		IF iObjState = 1 THEN																							// Objekt wurde geresettet
			iSkillCommand := 0;																								// Zurücksetzen von Command
			bDone := FALSE;																									// Zurücksetzen von Skill
			bSkillFertig := TRUE;									
		END_IF
			
		//  TRANSITION
		IF bSkillFertig THEN
			bSkillFertig := FALSE;																																											// Resetten von Objekt
			iState := 0;
		END_IF
		
// _________________________________________________________________________________________________________________________
3: 	// FEHLER
		// DO 	
		iSkillCommand := 0;
		
		bDone := FALSE;
		bBusy := FALSE;
		
		// TRANSITION
		IF bResetten THEN
			iState := 0;
		END_IF
		
// _________________________________________________________________________________________________________________________			
4: 	// LIMIT
		// DO 
		iSkillCommand := 0;
		bLimit := TRUE;																									// Limit wurde erreicht
		
		iSkillCommand := 3;																								// Objekt resetten
		
		IF iObjState = 1 THEN																							// Objekt wurde geresettet
			iSkillCommand := 0;																								// Zurücksetzen von Command
			bDone := FALSE;																									// Zurücksetzen von Skill
			bResetten := TRUE;								
		END_IF
	
		// TRANSITION
		IF bResetten THEN
			bResetten := FALSE;
			bLimit := FALSE;																							// Zurücksetzen von Output-Variable
			iSkillCommand := 3;																							// Resetten von Objekt 
			iState := 0;
		END_IF
			
// _________________________________________________________________________________________________________________________
5: 	// ERREICHT		
		// DO 
		iSkillCommand := 0;
		bDone := TRUE;																									// Skill wurde erfolgreich ausgeführt
		
		iSkillCommand := 3;																								// Objekt resetten
		
		IF iObjState = 1 THEN																							// Objekt wurde geresettet
			iSkillCommand := 0;																								// Zurücksetzen von Command
			bDone := FALSE;																									// Zurücksetzen von Skill
			bSkillFertig := TRUE;									
		END_IF
		
		// TRANSITION
		IF bSkillFertig THEN
			bSkillFertig := FALSE;
			iState := 0;
		END_IF
		
END_CASE

END_FUNCTION_BLOCK

// ---- POUs/01_Prozessmodell/02_Sequenzen/Seq_1.TcPOU
FUNCTION_BLOCK Seq_1
VAR_INPUT
	// Basis-Inputs
	bExecute			:BOOL;				// Trigger für Ausführung von Sequenz
	iSysCommand			:eSystemCommand;	// Steuerungsvariabel von System (Resetten)
	iSysState			:eSystemState;		// Information über Zustand von System
	
	
	// Prozess-Inputs 
	Position_1			:sRoboterProzessVariablen;
	Position_DOWN		:sRoboterProzessVariablen;
	Position_UP			:sRoboterProzessVariablen;
	Position_2			:sRoboterProzessVariablen;
END_VAR
VAR_OUTPUT
	bDone				:BOOL;				// Information ob Sequenz ausgfeührt wurde
	bBusy				:BOOL;				// Information ob Sequenz im Moment ausgeführt wird
	bError				:BOOL;				// Information ob sich Sequenz in Fehlerzustand befindet
END_VAR
VAR
	// Sequenz-Zustände
	iState				:eSequenceState;
	
	// Startvariablen (FB soll nur bei einer steigenden Flanke gestartet werden)
	fTrigger			:R_TRIG;			// Erkennung einer steigenden Flanke für den Starte
	fSwitch				:SR;				// Setzen des Signals
	bSwitchResett		:BOOL;				// Resetten des Signals
	
	// Zustandsvariablen
	bStarten			:BOOL;
	bStoppen			:BOOL;
	bResetten			:BOOL;
	
	// Management-Variablen:
	bFinished			:BOOL;
	bInit				:BOOL;
	
	// Skill-Instanziierungen
	P2P_Bewegung		:Skill_Position_anfahren;
	Position			:sRoboterProzessVariablen;
	
END_VAR

// Aufrufen von Skills und Ablauf
Ablauf();	
Skills();

//_______________________________________________________________
// Reaktion auf Fehler
IF bError THEN
	iState := 3;
END_IF	

// Reaktion auf Input-Variablen: 
	// Starten
	fTrigger(CLK := bExecute);
	fSwitch(Set1 := fTrigger.Q);
	
	IF fSwitch.Q1 THEN
		bStarten := TRUE;
	ELSE
		bStarten := FALSE;
	END_IF
	
	// Stoppen
	IF iSysCommand = 3 THEN
		bStoppen := TRUE;	
	ELSE 
		bStoppen := FALSE;	
	END_IF
	
	// Stoppen
	IF iSysCommand = 4 THEN
		bResetten := TRUE;	
	ELSE 
		bResetten := FALSE;	
	END_IF



//_______________________________________________________________
// Zustandsmanagement
CASE iState OF 
	0:	// BEREIT
			// DO	
			fSwitch.RESET := FALSE;
				
			// TRANSITION
			IF bStarten THEN
				fSwitch.RESET := TRUE;
				iState := 1;																							// Starten des Objektes 
			END_IF
	// ________________________________________________________________________________			
	1:	// LAUFEND
			// DO
			bBusy := TRUE;	

			IF bStoppen THEN
				SFCReset := TRUE;
				bBusy := FALSE;
			END_IF	
			
			// TRANSITION
			IF bFinished THEN
				bFinished := FALSE;
				bBusy := FALSE;
				iState := 2;
			END_IF
			
			IF bInit THEN
				bInit := FALSE;
				SFCReset := FALSE;
				iState := 0;
			END_IF

	// ________________________________________________________________________________					
	2:	// ABGESCHLOSSEN
			// DO
			bDone := TRUE;			
						
			// TRANSITION
			IF bDone THEN
				bDone := FALSE;
				iState := 0;
			END_IF
	// ________________________________________________________________________________					
	3:	// FEHLER
			// DO
			bDone := FALSE;
			bBusy := FALSE;
			
			// TRANSITION
			IF bResetten THEN
				bError := FALSE;
				iState := 0;
			END_IF
			
END_CASE

ACTION Ablauf:
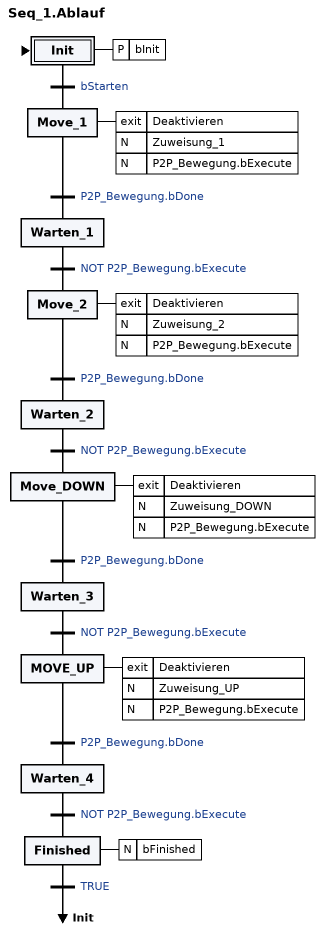
INITIAL_STEP Init:
    bInit(P);
END_STEP
TRANSITION FROM Init TO Move_1
    := bStarten;
END_TRANSITION
STEP Move_1:
    Deaktivieren(P0);  // exit action
    Zuweisung_1(N);
    P2P_Bewegung.bExecute(N);
END_STEP
TRANSITION FROM Move_1 TO Warten_1
    := P2P_Bewegung.bDone;
END_TRANSITION
STEP Warten_1:
END_STEP
TRANSITION FROM Warten_1 TO Move_2
    := NOT P2P_Bewegung.bExecute;
END_TRANSITION
STEP Move_2:
    Deaktivieren(P0);  // exit action
    Zuweisung_2(N);
    P2P_Bewegung.bExecute(N);
END_STEP
TRANSITION FROM Move_2 TO Warten_2
    := P2P_Bewegung.bDone;
END_TRANSITION
STEP Warten_2:
END_STEP
TRANSITION FROM Warten_2 TO Move_DOWN
    := NOT P2P_Bewegung.bExecute;
END_TRANSITION
STEP Move_DOWN:
    Deaktivieren(P0);  // exit action
    Zuweisung_DOWN(N);
    P2P_Bewegung.bExecute(N);
END_STEP
TRANSITION FROM Move_DOWN TO Warten_3
    := P2P_Bewegung.bDone;
END_TRANSITION
STEP Warten_3:
END_STEP
TRANSITION FROM Warten_3 TO MOVE_UP
    := NOT P2P_Bewegung.bExecute;
END_TRANSITION
STEP MOVE_UP:
    Deaktivieren(P0);  // exit action
    Zuweisung_UP(N);
    P2P_Bewegung.bExecute(N);
END_STEP
TRANSITION FROM MOVE_UP TO Warten_4
    := P2P_Bewegung.bDone;
END_TRANSITION
STEP Warten_4:
END_STEP
TRANSITION FROM Warten_4 TO Finished
    := NOT P2P_Bewegung.bExecute;
END_TRANSITION
STEP Finished:
    bFinished(N);
END_STEP
TRANSITION FROM Finished TO Init
    := TRUE;
END_TRANSITION
END_ACTION

ACTION Deaktivieren:
P2P_Bewegung.bExecute := FALSE;
END_ACTION

ACTION Skills:
P2P_Bewegung(
    iSysCommand := GVL.SystemCommand,
    iObjState := Anlage.UR5.P_State,
    iSysState := GVL.SystemState,
    sProzessvariablen := Position); // Skill_Position_anfahren
Anlage.UR5.Prozessvariablen := P2P_Bewegung.sObjektvariablen;
Anlage.UR5.iSkillCommand_1 := P2P_Bewegung.iSkillCommand;
END_ACTION

ACTION Zuweisung_1:
Position := Position_1;
END_ACTION

ACTION Zuweisung_2:
Position := Position_2;
END_ACTION

ACTION Zuweisung_DOWN:
Position := Position_DOWN;
END_ACTION

ACTION Zuweisung_UP:
Position := Position_UP;
END_ACTION

END_FUNCTION_BLOCK

// ---- POUs/02_Anlagenmodell/02_Objektklassen/00_Referenz/Basis_Objekt.TcPOU
FUNCTION_BLOCK Basis_Objekt EXTENDS GrundstrukturObjekt
VAR_INPUT
END_VAR
VAR_OUTPUT
END_VAR
VAR
END_VAR

// Instanziierungen
	
//____________________________________________________________________________________________
// Input-Command-Verwaltung
	// System
	IF iSysCommand = 2 AND iState = 0 THEN			// Objekt einschalten
		bEinschalten := TRUE;
	ELSE 
		bEinschalten := FALSE;
	END_IF
	
	IF iSysCommand = 1 AND iState = 1 THEN			// Objekt ausschalten
		bAusschalten := TRUE;		
	ELSE 
		bAusschalten := FALSE;		
	END_IF
	
	IF iSysCommand = 3 THEN							// Objekt beendet Prozess
		bStoppen := TRUE;
	ELSE
		bStoppen := FALSE;
	END_IF
	
	IF iSysCommand = 4 THEN							// System resettet Objekt
		bResettenSystem := TRUE;
	ELSE
		bResettenSystem := FALSE;
	END_IF
	
	// Skill
	IF iSkillCommand_1 = 1 THEN						// Skill startet Prozess
		bStarten := TRUE;
	ELSE 
		bStarten := FALSE;
	END_IF
	
	IF iSkillCommand_1 = 2 THEN						// Skill beendet Prozess
		bSkillFertig := TRUE;
	ELSE
		bSkillFertig := FALSE;
	END_IF
	
	IF iSkillCommand_1 = 3 THEN						// Skill resettet Objekt
 		bResettenSkill := TRUE;
	ELSE
		bResettenSkill := FALSE;
	END_IF

//____________________________________________________________________________________________
// Interner Methodenaufruf (Durch System oder Skill)

//____________________________________________________________________________________________
// Datenerfassungsprozess

//____________________________________________________________________________________________
// Zustandsmanagement

IF bFehler THEN 
	iState := 7;
END_IF

CASE iState OF 
	0: // AUS
		// DO
		
		// TRANSITION
			IF bEinschalten THEN																	// Verbindung wird aufgebaut
				iState := 1;
			END_IF
			
	//____________________________________________________________________________________________
	1: // BEREIT
		// DO

		// TRANSITION
																									// Manuell-Modus wird eingeschalten
													
			 IF bStarten THEN																		// Objekt führt Prozessdurch
				 iState := 3;
			 END_IF			
	//____________________________________________________________________________________________
	2: // MANUELL
		// DO
		
		// TRANSITION
	
	//____________________________________________________________________________________________
	3: // LAUFEND
		// DO
		
		// TRANSITION
			IF bObjektFertig THEN
				bObjektFertig := FALSE;
				iState := 4;
			END_IF
			
			IF bStoppen THEN	
				
				IF bSkillFertig THEN
					iState := 5;
				END_IF
					
				IF bStoppen THEN
					iState := 6;
				END_IF
					
			END_IF
	
	//____________________________________________________________________________________________
	4: // ABGESCHLOSSEN_INTERN
		// DO
		
		// TRANSITION
			IF bResettenSkill THEN																	// Objekt resetten		
				iState := 1;
			END_IF
	//____________________________________________________________________________________________
	5: // ABGESCHLOSSEN_EXTERN
		// DO																					
		
		// TRANSITION
			IF bResettenSkill THEN																	// Objekt resetten
				iState := 1;
			END_IF
	
	//____________________________________________________________________________________________
	6: // GESTOPPT
		// DO
		
		// TRANSITION
			IF bResettenSystem THEN																	// Objekt resetten
				iState := 1;
			END_IF
	
	//____________________________________________________________________________________________
	7: // FEHLER
		// DO
			bError := bFehler;
			
		// TRANSITION
			IF bResettenSystem THEN																	// Objekt resetten
				bFehler	 := FALSE;
				bError := FALSE;
				iState := 1;
			END_IF
	
END_CASE

END_FUNCTION_BLOCK

// ---- GlobalTextList.TcGTLO
TEXTLIST GlobalTextList
  425 = '%s'
  484 = 'AKTIVIEREN'
  874 = 'AUSCHALTEN'
  468 = 'EINSCHALTEN'
  440 = 'EXECUTE'
  917 = 'Greifer_Test'
  764 = 'KEINE'
  545 = 'ObjectState'
  207 = 'Position anfahren'
  913 = 'Position anfahren:'
  462 = 'RES PROZESS'
  680 = 'RES PROZESSET'
  988 = 'RESET'
  482 = 'RESET Prozess¨'
  303 = 'RESETTEN'
  707 = 'SkillCommand'
  512 = 'SkillState'
  844 = 'START'
  554 = 'STARTEN'
  351 = 'STOPPEN'
  785 = 'SystemCommand'
  668 = 'Test-Steuerung'
  54 = 'UR5:'
END_TEXTLIST

// ---- VISUs/00_Debug/SystemState.TcVIS
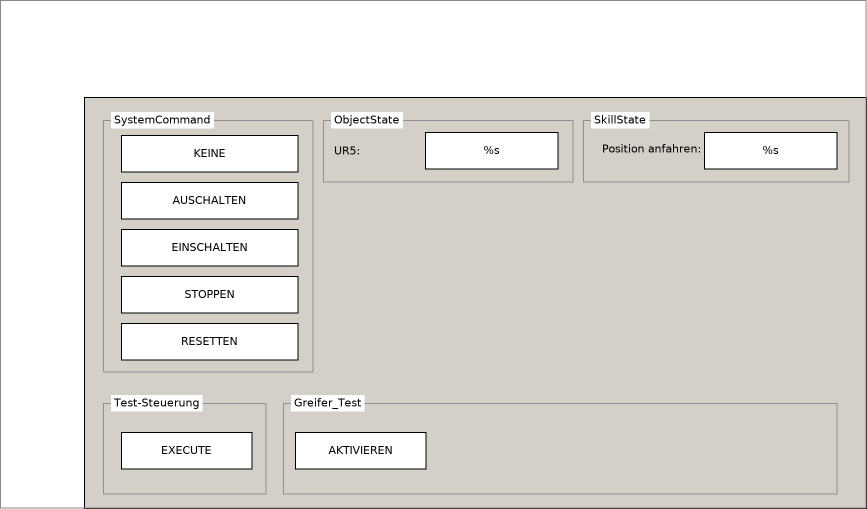
VISUALIZATION SystemState  // 867x509
    RoundedRectangle (84,97 783x412)
    GroupBox (103,112 210x260), "SystemCommand"
        RoundedRectangle (18,70 177x37), "AUSCHALTEN"
            OnMouseClick: execute { GVL.SystemCommand := 1; }
        RoundedRectangle (18,117 177x37), "EINSCHALTEN"
            OnMouseClick: execute { GVL.SystemCommand := 2; }
        RoundedRectangle (18,164 177x37), "STOPPEN"
            OnMouseClick: execute { GVL.SystemCommand := 3; }
        RoundedRectangle (18,211 177x37), "RESETTEN"
            OnMouseClick: execute { GVL.SystemCommand := 4; }
        RoundedRectangle (18,23 177x37), "KEINE"
            OnMouseClick: execute { GVL.SystemCommand := 0; }
    GroupBox (323,112 250x70), "ObjectState"
        RoundedRectangle (102,20 133x37), "%s", text variable: Anlage.UR5.P_State, input disabled if: TRUE
        Label (8,24 38x30), "UR5:"
    GroupBox (583,112 266x70), "SkillState"
        RoundedRectangle (121,20 133x37), "%s", input disabled if: TRUE
        Label (16,22 110x30), "Position anfahren:"
    GroupBox (103,395 163x99), "Test-Steuerung"
        RoundedRectangle (18,37 131x37), "EXECUTE"
            tap MAIN.Execute
    GroupBox (283,395 554x99), "Greifer_Test"
        RoundedRectangle (12,37 131x37), "AKTIVIEREN"
            OnMouseClick: execute { Anlage.Gripper.Aktivieren(); }
END_VISUALIZATION
